// TIA Portal V17 export
// export: Created 2026-04-13T11:12:42.1292007Z, ExportSetting WithDefaults, DisplayName Totally Integrated Automation Portal, DisplayVersion V17 Update 4, DisplayName TIA Portal Openness, DisplayVersion V17 Update 4, DisplayName TIA Portal Version Control Interface, DisplayVersion V17, DisplayName SINAMICS Startdrive Advanced, DisplayVersion V17, DisplayName SINAMICS Startdrive G130, G150, S120, S150, SINAMICS MV, S210, DisplayVersion V17, DisplayName SINAMICS Startdrive G110M, G120, G120C, G120D, G120P, G115D, DisplayVersion V17, DisplayName STEP 7 Professional, DisplayVersion V17 Update 4, DisplayName STEP 7 Safety, DisplayVersion V17, DisplayName WinCC Professional, DisplayVersion V17 Update 4
FUNCTION_BLOCK "步模式"   // FB60, SCL
{ S7_Optimized_Access := 'TRUE' }
VERSION : 0.1
// stored: AutoNumber true, IsIECCheckEnabled false, IsRetainMemResEnabled false, MemoryReserve 100, SetENOAutomatically false, UDAEnableTagReadback false
   VAR_INPUT
      FK : Bool;   // 动作反馈
   END_VAR
   VAR_IN_OUT
      IN : Bool;   // 进入步段条件
      RUN : Bool;   // 动作运行,运行完后就关闭,一般接TON
      DONE : Bool;   // 动作完成,一般是一个标注位
      OVER : Bool;   // 步段完成,运行完之后继续开状态
   END_VAR
BEGIN
   #OVER := #IN AND (#DONE OR #OVER);
   #RUN := #IN AND NOT #OVER ;
   #DONE := #RUN AND #FK;
END_FUNCTION_BLOCK
